// TIA Portal V19 export
TYPE "RecordData"
   STRUCT
      "b" : Array[0..231] of Byte;
   END_STRUCT;
END_TYPE
